% RSLogix 500 project AnalogVALVE-PUMP_BAK001.RSS, saved by version 8.30.00.16 %
PROJECT "UNTITLED"    % processor: Bul.1763 MicroLogix 1100 Series B %

PROGRAM FILES
  LAD 2 "MAIN"  3 rungs
  LAD 4 "DIGITAL IO"  6 rungs
  LAD 5 "CONTROLS"  6 rungs

DATA FILES
  O0 OUTPUT  5 elements
  I1 INPUT  14 elements
  S2 STATUS  66 elements
  B3 BINARY  1 elements
  T4 TIMER  2 elements
  C5 COUNTER  1 elements
  R6 CONTROL  1 elements
  N7 INTEGER  1 elements
  F8 FLOAT  1 elements

LADDER 2 "MAIN"
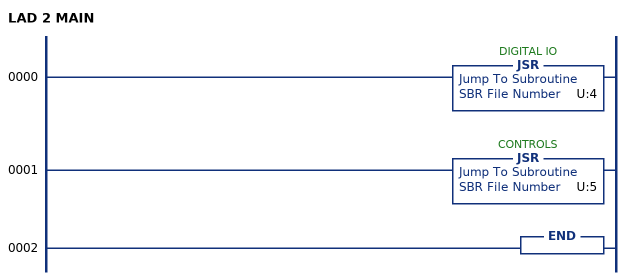
% Rung: 0 %
SOR JSR U:4 EOR
%   U:4  "DIGITAL IO" %
% Rung: 1 %
SOR JSR U:5 EOR
%   U:5  "CONTROLS" %
% Rung: 2 %
SOR END EOR

LADDER 4 "DIGITAL IO"
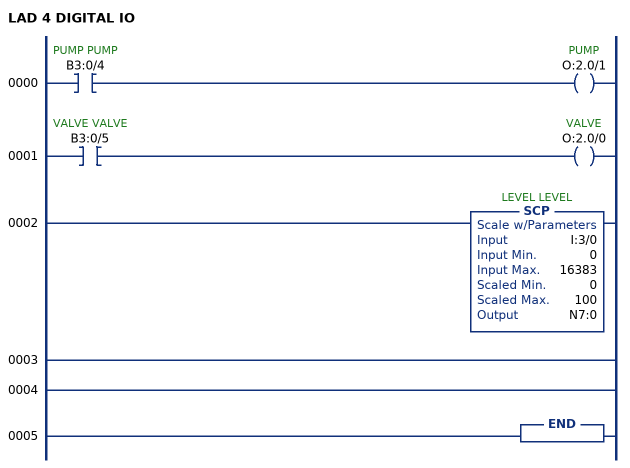
% Rung: 0 %
SOR XIC B3:0/4 OTE O:2.0/1 EOR
%   B3:0/4  PUMP  "PUMP" %
%   O:2.0/1  "PUMP" %
% Rung: 1 %
SOR XIC B3:0/5 OTE O:2.0/0 EOR
%   B3:0/5  VALVE  "VALVE" %
%   O:2.0/0  "VALVE" %
% Rung: 2 %  % edit flag set %
SOR SCP I:3/0 0 16383 0 100 N7:0 EOR
%   N7:0  LEVEL  "LEVEL" %
% Rung: 3 %  % edit flag set %
SOR EOR
% Rung: 4 %  % edit flag set %
SOR EOR
% Rung: 5 %
SOR END EOR

LADDER 5 "CONTROLS"
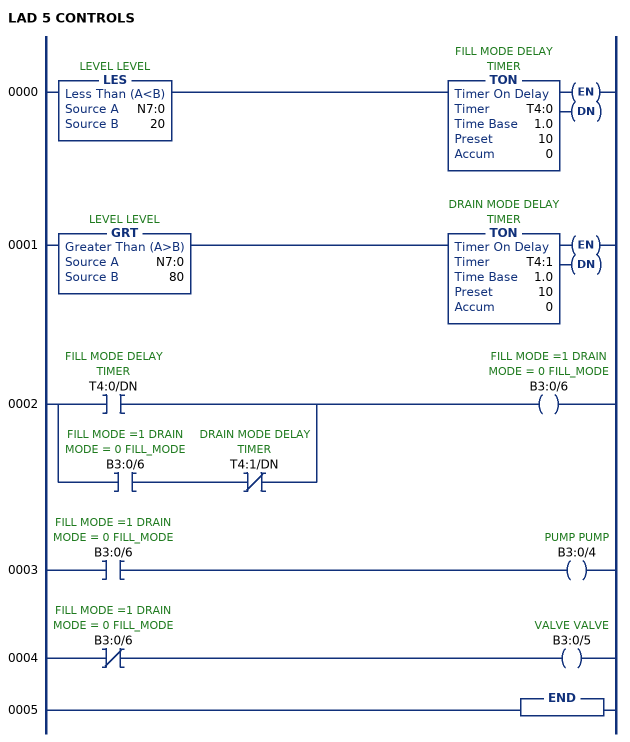
% Rung: 0 %  % edit flag set %
SOR LES N7:0 20 TON T4:0 1.0 10 0 EOR
%   N7:0  LEVEL  "LEVEL" %
%   T4:0  "FILL MODE DELAY TIMER" %
% Rung: 1 %  % edit flag set %
SOR GRT N7:0 80 TON T4:1 1.0 10 0 EOR
%   N7:0  LEVEL  "LEVEL" %
%   T4:1  "DRAIN MODE DELAY TIMER" %
% Rung: 2 %
SOR BST XIC T4:0/DN NXB XIC B3:0/6 XIO T4:1/DN BND OTE B3:0/6 EOR
%   T4:0/DN  "FILL MODE DELAY TIMER" %
%   B3:0/6  FILL_MODE  "FILL MODE =1 DRAIN MODE = 0" %
%   T4:1/DN  "DRAIN MODE DELAY TIMER" %
% Rung: 3 %
SOR XIC B3:0/6 OTE B3:0/4 EOR
%   B3:0/6  FILL_MODE  "FILL MODE =1 DRAIN MODE = 0" %
%   B3:0/4  PUMP  "PUMP" %
% Rung: 4 %
SOR XIO B3:0/6 OTE B3:0/5 EOR
%   B3:0/6  FILL_MODE  "FILL MODE =1 DRAIN MODE = 0" %
%   B3:0/5  VALVE  "VALVE" %
% Rung: 5 %
SOR END EOR

OTHER DOCUMENTED ADDRESSES
  B3:0/0  LL_SWITCH  "LL SWITCH"
  B3:0/1  L_SWITCH  "L SWITCH"
  B3:0/2  H_SWITCH  "H SWITCH"
  B3:0/3  HH_SWITCH  "HH SWITCH"
  I:0.0/0  "LL SWITCH INPUT"
  I:0.0/1  "L SWITCH INPUT"
  I:0.0/2  "H SWITCH INPUT"
  I:0.0/3  "HH SWITCH INPUT"
  I:3.0/0  "LEVEL SENSOR INPUT"

DATA TABLE (non-zero values as saved)
DATA T4
% .PRE .ACC %
% T4:0 % 10 0
% T4:1 % 10 0
